FUNCTION_BLOCK FB_ModbusCon
VAR_INPUT
    bEnable: BOOL;
END_VAR
VAR_OUTPUT
    // Operating data from inverter
    stInverter: ST_OpDataInverter;
    // Operating data from meter
    stMeter: ST_OpDataMeter;
    // Operating data from storage
    stStorage: ST_OpDataStorage;
    // Connection is ready and not locked out
    bReady: BOOL;
END_VAR
VAR
    // IP address of the target device
    {attribute 'hide'}
    _sInverterIPAddr: STRING;
    // Port number of the target device
    {attribute 'hide'}
    _nInverterTCPPort: UINT;
    // Modbus RTU ID of inverter, value must be 16#FF if addressed directly via TCP/IP
    {attribute 'hide'}
    _nInverterUnitID: BYTE;
    // Modbus RTU ID of meter, value must be 16#FF if addressed directly via TCP/IP
    {attribute 'hide'}
    _nMeterUnitID: BYTE;
    // Timeout that may not be exceeded by execution of the ADS command
    {attribute 'hide'}
    _tConnectionTimeout: TIME;
    // Timeout between modbus commands sent to target device
    {attribute 'hide'}
    _tConnectionCoolDown: TIME;

    // Modbus connection to read registers
    fbReadRegister: FB_MBReadRegs;
    // Connection cooldown timeout between requests
    fbConnectionCoolDown: TOF;

    // Register data of inverter
    stInverterRegisterData: ST_RegMapInverter;
    // Register data of meter
    stMeterRegisterData: ST_RegMapMeter;
    // Register data of storage
    stStorageRegisterData: ST_RegMapStorage;

    // Number of current tried countermeasures after modbus connection error
    nConnectionCountermeasure: INT;
    // Number of current tried countermeasures after modbus request error regarding inverter
    nInverterCountermeasure: INT;
    // Number of current tried countermeasures after modbus request error regarding meter
    nMeterCountermeasure: INT;
    // Number of current tried countermeasures after modbus request error regarding storage
    nStorageCountermeasure: INT;

    // Current state of modbus read registers
    eReadState: (WAIT_FOR_ENABLE, PREPARE_READ_REGS, EXECUTE_READ_REGS, WAIT_READ_REGS_FEEDBACK, ASSIGN_VALUES, SELECT_NEXT_SUBSYTEM, CON_COOL_DOWN, CON_LOCKOUT);
    // Select subsystem for request to prevent parallel requests
    eCurrentSubsystem: (INVERTER, METER, STORAGE);

    // Show only events with minimum severety level
    {attribute 'hide'}
    _eTraceLevel: TcEventSeverity := TcEventSeverity.Warning;

    fbAlarmMbConnectionError: FB_TcAlarm;
    fbAlarmMbFunctionInverterError: FB_TcAlarm;
    fbAlarmMbFunctionMeterError: FB_TcAlarm;
    fbAlarmMbFunctionStorageError: FB_TcAlarm;
    fbAlarmMbConnectionLocked: FB_TcAlarm;
    fbMessageMbOpDataIsUpdated: FB_TcMessage;
    fbMessageMbUncatchedError: FB_TcMessage;
    fbMessageMbReceivedBytesMismatch: FB_TcMessage;
END_VAR
VAR CONSTANT
    // Number of output registers used by stInverterRegisterData
    nInverterRegQuantity: WORD := 16;
    // Start address of the output register used by stInverterRegisterData
    nInverterMBStartAddr: WORD := 40071;
    // Number of output registers used by stMeterRegisterData
    nMeterRegQuantity: WORD := 21;
    // Start address of the output register used by stMeterRegisterData
    nMeterMBStartAddr: WORD := 40071;
    // Number of output registers used by stStorageRegisterData
    nStorageRegQuantity: WORD := 4;
    // Start address of the output register used by stStorageRegisterData
    nStorageMBStartAddr: WORD := 40351;
    // Number of attempted countermeasures before connection lockout (connection error)
    nConnectionCmBeforeLockout: INT := 5;
    // Number of attempted countermeasures before connection lockout (subsystem error)
    nSubsystemCmBeforeLockout: INT := 2;
END_VAR

fbReadRegister(sIPAddr := sInverterIPAddr, nTCPPort := nInverterTCPPort, tTimeout := tConnectionTimeout);
fbConnectionCoolDown();

// Set ready state
bReady := eReadState <> CON_LOCKOUT;

// Default operating data has not been updated this cycle
stInverter.bOpDataIsUpdated := FALSE;
stMeter.bOpDataIsUpdated := FALSE;
stStorage.bOpDataIsUpdated := FALSE;

// State machine
CASE eReadState OF
    WAIT_FOR_ENABLE:
        IF bEnable AND fbConnectionCoolDown.Q THEN
            eReadState := CON_COOL_DOWN;
        ELSIF bEnable THEN
            eReadState := PREPARE_READ_REGS;
        END_IF

    PREPARE_READ_REGS:
        CASE eCurrentSubsystem OF
            INVERTER:
                fbReadRegister.nUnitID := nInverterUnitID;
                fbReadRegister.nQuantity := nInverterRegQuantity;
                fbReadRegister.nMBAddr := nInverterMBStartAddr;
                fbReadRegister.cbLength := SIZEOF(stInverterRegisterData);
                fbReadRegister.pDestAddr := ADR(stInverterRegisterData);

            METER:
                fbReadRegister.nUnitID := nMeterUnitID;
                fbReadRegister.nQuantity := nMeterRegQuantity;
                fbReadRegister.nMBAddr := nMeterMBStartAddr;
                fbReadRegister.cbLength := SIZEOF(stMeterRegisterData);
                fbReadRegister.pDestAddr := ADR(stMeterRegisterData);

            STORAGE:
                fbReadRegister.nUnitID := nInverterUnitID;
                fbReadRegister.nQuantity := nStorageRegQuantity;
                fbReadRegister.nMBAddr := nStorageMBStartAddr;
                fbReadRegister.cbLength := SIZEOF(stStorageRegisterData) - 2;
                fbReadRegister.pDestAddr := ADR(stStorageRegisterData);
        END_CASE

        eReadState := EXECUTE_READ_REGS;

    EXECUTE_READ_REGS:
        fbReadRegister.bExecute := TRUE;
        fbConnectionCoolDown.IN := TRUE;
        eReadState := WAIT_READ_REGS_FEEDBACK;

    WAIT_READ_REGS_FEEDBACK:
        fbReadRegister.bExecute := FALSE;
        IF NOT fbReadRegister.bBusy THEN
            fbConnectionCoolDown.IN := FALSE;
            ConnectionErrorHandler();

            IF ConnectionLockoutIsActive() THEN
                // Lockout modbus connection
                eReadState := CON_LOCKOUT;
            ELSIF fbReadRegister.cbLength <> fbReadRegister.cbRead THEN
                // Send message M_MbReceivedBytesMismatch
                IF fbMessageMbReceivedBytesMismatch.eSeverity >= eTraceLevel THEN
                    fbMessageMbReceivedBytesMismatch.ipArguments.Clear();
                    fbMessageMbReceivedBytesMismatch.ipArguments.AddBool(value := eCurrentSubsystem = INVERTER);
                    fbMessageMbReceivedBytesMismatch.ipArguments.AddBool(value := eCurrentSubsystem = METER);
                    fbMessageMbReceivedBytesMismatch.ipArguments.AddBool(value := eCurrentSubsystem = STORAGE);
                    fbMessageMbReceivedBytesMismatch.Send();
                END_IF
                // Skip assigning values to output variable
                eReadState := SELECT_NEXT_SUBSYTEM;
            ELSE
                eReadState := ASSIGN_VALUES;
            END_IF
        END_IF

    ASSIGN_VALUES:
        CASE eCurrentSubsystem OF
            INVERTER:
                stInverter.bOpDataIsUpdated := TRUE;
                stInverter.fCurrentL1 := Scale(stInverterRegisterData.nCurrentL1, stInverterRegisterData.nSfCurrent);
                stInverter.fCurrentL2 := Scale(stInverterRegisterData.nCurrentL2, stInverterRegisterData.nSfCurrent);
                stInverter.fCurrentL3 := Scale(stInverterRegisterData.nCurrentL3, stInverterRegisterData.nSfCurrent);
                stInverter.fVoltageL1L2 := Scale(stInverterRegisterData.nVoltageL1L2, stInverterRegisterData.nSfVoltage);
                stInverter.fVoltageL2L3 := Scale(stInverterRegisterData.nVoltageL2L3, stInverterRegisterData.nSfVoltage);
                stInverter.fVoltageL3L1 := Scale(stInverterRegisterData.nVoltageL3L1, stInverterRegisterData.nSfVoltage);
                stInverter.fVoltageL1N := Scale(stInverterRegisterData.nVoltageL1N, stInverterRegisterData.nSfVoltage);
                stInverter.fVoltageL2N := Scale(stInverterRegisterData.nVoltageL2N, stInverterRegisterData.nSfVoltage);
                stInverter.fVoltageL3N := Scale(stInverterRegisterData.nVoltageL3N, stInverterRegisterData.nSfVoltage);
                stInverter.fPower := Scale(stInverterRegisterData.nPower, stInverterRegisterData.nSfPower);
                stInverter.fFrequency := Scale(stInverterRegisterData.nFrequency, stInverterRegisterData.nSfFrequency);

            METER:
                stMeter.bOpDataIsUpdated := TRUE;
                stMeter.fCurrentL1 := Scale(stMeterRegisterData.nCurrentL1, stMeterRegisterData.nSfCurrent);
                stMeter.fCurrentL2 := Scale(stMeterRegisterData.nCurrentL2, stMeterRegisterData.nSfCurrent);
                stMeter.fCurrentL3 := Scale(stMeterRegisterData.nCurrentL3, stMeterRegisterData.nSfCurrent);
                stMeter.fVoltageL1L2 := Scale(stMeterRegisterData.nVoltageL1L2, stMeterRegisterData.nSfVoltage);
                stMeter.fVoltageL2L3 := Scale(stMeterRegisterData.nVoltageL2L3, stMeterRegisterData.nSfVoltage);
                stMeter.fVoltageL3L1 := Scale(stMeterRegisterData.nVoltageL3L1, stMeterRegisterData.nSfVoltage);
                stMeter.fVoltageL1N := Scale(stMeterRegisterData.nVoltageL1N, stMeterRegisterData.nSfVoltage);
                stMeter.fVoltageL2N := Scale(stMeterRegisterData.nVoltageL2N, stMeterRegisterData.nSfVoltage);
                stMeter.fVoltageL3N := Scale(stMeterRegisterData.nVoltageL3N, stMeterRegisterData.nSfVoltage);
                stMeter.fPower := Scale(stMeterRegisterData.nPower, stMeterRegisterData.nSfPower);
                stMeter.fPowerL1 := Scale(stMeterRegisterData.nPowerL1, stMeterRegisterData.nSfPower) - 100;
                stMeter.fPowerL2 := Scale(stMeterRegisterData.nPowerL2, stMeterRegisterData.nSfPower) - 100;
                stMeter.fPowerL3 := Scale(stMeterRegisterData.nPowerL3, stMeterRegisterData.nSfPower) - 100;
                stMeter.fFrequency := Scale(stMeterRegisterData.nFrequency, stMeterRegisterData.nSfFrequency);

            STORAGE:
                stStorage.bOpDataIsUpdated := TRUE;
                stStorage.nStateOfCharge := REAL_TO_INT(Scale(stStorageRegisterData.nStateOfCharge, stStorageRegisterData.nSfStateOfCharge));
                stStorage.eState := stStorageRegisterData.nState;
        END_CASE
        eReadState := SELECT_NEXT_SUBSYTEM;

        // Send message M_MbOpDataIsUpdated
        IF fbMessageMbOpDataIsUpdated.eSeverity >= eTraceLevel THEN
            fbMessageMbOpDataIsUpdated.ipArguments.Clear();
            fbMessageMbOpDataIsUpdated.ipArguments.AddBool(value := stInverter.bOpDataIsUpdated);
            fbMessageMbOpDataIsUpdated.ipArguments.AddBool(value := stMeter.bOpDataIsUpdated);
            fbMessageMbOpDataIsUpdated.ipArguments.AddBool(value := stStorage.bOpDataIsUpdated);
            fbMessageMbOpDataIsUpdated.Send();
        END_IF

    SELECT_NEXT_SUBSYTEM:
        CASE eCurrentSubsystem OF
            INVERTER:
                eCurrentSubsystem := METER;

            METER:
                eCurrentSubsystem := STORAGE;

            STORAGE:
                eCurrentSubsystem := INVERTER;

            ELSE
                eCurrentSubsystem := INVERTER;
        END_CASE
        eReadState := CON_COOL_DOWN;

    CON_COOL_DOWN:
        IF NOT bEnable THEN
            eReadState := WAIT_FOR_ENABLE;
        END_IF

        IF NOT fbConnectionCoolDown.Q THEN
            eReadState := PREPARE_READ_REGS;
        END_IF

    CON_LOCKOUT:
        (* Perform reset using Reset() function *)
END_CASE

METHOD PRIVATE ConnectionErrorHandler
IF ConnectionLockoutIsActive() THEN
    RETURN;
END_IF

IF fbReadRegister.bError THEN
    // Apply countermeasure if ADS error occured
    CASE fbReadRegister.nErrId OF
        16#8001, // Modbus function not implemented
        16#8002, // Invalid address or length
        16#8003, // Invalid parameters: incorrect number of registers
        16#8004: // Modbus server error
            CASE eCurrentSubsystem OF
                INVERTER:
                    nInverterCountermeasure := nInverterCountermeasure + 1;
                METER:
                    nMeterCountermeasure := nMeterCountermeasure + 1;
                STORAGE:
                    nStorageCountermeasure := nStorageCountermeasure + 1;
            END_CASE
            

        Global.E_TcSystemEventClass.TCPSendError, // TCP send error
        Tc2_System.E_AdsErr.CLIENT_SYNCTIMEOUT:   // Remote terminal is not responding in the specified ADS timeout
            nConnectionCountermeasure := nConnectionCountermeasure + 1;
            fbConnectionCoolDown.PT := tConnectionCoolDown + tConnectionCoolDown * LREAL_TO_INT(EXPT(nConnectionCountermeasure, 2));

        ELSE
            // Send message M_MbUncatchedError
            IF fbMessageMbUncatchedError.eSeverity >= eTraceLevel THEN
                fbMessageMbUncatchedError.ipArguments.Clear();
                fbMessageMbUncatchedError.ipArguments.AddUDInt(value := fbReadRegister.nErrId);
                fbMessageMbUncatchedError.Send();
            END_IF
    END_CASE

ELSE
    // Defer possibly still active countermeasure
    nInverterCountermeasure := 0;
    nMeterCountermeasure := 0;
    nStorageCountermeasure := 0;
    nConnectionCountermeasure := 0;

    // Reset connection cooldown timeout
    fbConnectionCoolDown.PT := tConnectionCoolDown;
END_IF

IF nConnectionCountermeasure > 0 AND fbAlarmMbConnectionError.eSeverity >= eTraceLevel AND NOT fbAlarmMbConnectionError.bRaised THEN
    // Raise alarm F_MbConnectionError
    fbAlarmMbConnectionError.ipArguments.AddUDInt(value := fbReadRegister.nErrId);
    fbAlarmMbConnectionError.Raise();
ELSIF nConnectionCountermeasure = 0 AND fbAlarmMbConnectionError.bRaised THEN
    // Clear alarm F_MbConnectionError
    fbAlarmMbConnectionError.ipArguments.Clear();
    fbAlarmMbConnectionError.Clear();
END_IF

IF nInverterCountermeasure > 0 AND fbAlarmMbFunctionInverterError.eSeverity >= eTraceLevel AND NOT fbAlarmMbFunctionInverterError.bRaised THEN
    // Raise alarm F_MbFunctionInverterError
    fbAlarmMbFunctionInverterError.ipArguments.AddUDInt(value := fbReadRegister.nErrId);
    fbAlarmMbFunctionInverterError.Raise();
ELSIF nInverterCountermeasure = 0 AND fbAlarmMbFunctionInverterError.bRaised THEN
    // Clear alarm F_MbFunctionInverterError
    fbAlarmMbFunctionInverterError.ipArguments.Clear();
    fbAlarmMbFunctionInverterError.Clear();
END_IF

IF nMeterCountermeasure > 0 AND fbAlarmMbFunctionMeterError.eSeverity >= eTraceLevel AND NOT fbAlarmMbFunctionMeterError.bRaised THEN
    // Raise alarm F_MbFunctionMeterError
    fbAlarmMbFunctionMeterError.ipArguments.AddUDInt(value := fbReadRegister.nErrId);
    fbAlarmMbFunctionMeterError.Raise();
ELSIF nMeterCountermeasure = 0 AND fbAlarmMbFunctionMeterError.bRaised THEN
    // Clear alarm F_MbFunctionMeterError
    fbAlarmMbFunctionMeterError.ipArguments.Clear();
    fbAlarmMbFunctionMeterError.Clear();
END_IF

IF nStorageCountermeasure > 0 AND fbAlarmMbFunctionStorageError.eSeverity >= eTraceLevel AND NOT fbAlarmMbFunctionStorageError.bRaised THEN
    // Raise alarm F_MbFunctionStorageError
    fbAlarmMbFunctionStorageError.ipArguments.AddUDInt(value := fbReadRegister.nErrId);
    fbAlarmMbFunctionStorageError.Raise();
ELSIF nStorageCountermeasure = 0 AND fbAlarmMbFunctionStorageError.bRaised THEN
    // Clear alarm F_MbFunctionStorageError
    fbAlarmMbFunctionStorageError.ipArguments.Clear();
    fbAlarmMbFunctionStorageError.Clear();
END_IF
END_METHOD

METHOD PRIVATE ConnectionLockoutIsActive : BOOL
// Default to false, no lockout active
ConnectionLockoutIsActive := FALSE;

// Return if already in locked state
IF eReadState = CON_LOCKOUT THEN
    ConnectionLockoutIsActive := TRUE;
    RETURN;
END_IF

IF nConnectionCountermeasure > nConnectionCmBeforeLockout THEN
    ConnectionLockoutIsActive := TRUE;
    // Add reference to F_MbConnectionError as argument to F_MbConnectionLocked
    IF fbAlarmMbConnectionLocked.eSeverity >= eTraceLevel AND NOT fbAlarmMbConnectionLocked.bRaised THEN
        fbAlarmMbConnectionLocked.ipArguments.AddEventReferenceId(nEventId := fbAlarmMbConnectionError.nEventId);
    END_IF
END_IF

if nInverterCountermeasure > nSubsystemCmBeforeLockout THEN
    ConnectionLockoutIsActive := TRUE;
    // Add reference to F_MbFunctionInverterError as argument to F_MbConnectionLocked
    IF fbAlarmMbConnectionLocked.eSeverity >= eTraceLevel AND NOT fbAlarmMbConnectionLocked.bRaised THEN
        fbAlarmMbConnectionLocked.ipArguments.AddEventReferenceId(nEventId := fbAlarmMbFunctionInverterError.nEventId);
    END_IF
END_IF

if nMeterCountermeasure > nSubsystemCmBeforeLockout THEN
    ConnectionLockoutIsActive := TRUE;
    // Add reference to F_MbFunctionMeterError as argument to F_MbConnectionLocked
    IF fbAlarmMbConnectionLocked.eSeverity >= eTraceLevel AND NOT fbAlarmMbConnectionLocked.bRaised THEN
        fbAlarmMbConnectionLocked.ipArguments.AddEventReferenceId(nEventId := fbAlarmMbFunctionMeterError.nEventId);
    END_IF
END_IF

if nStorageCountermeasure > nSubsystemCmBeforeLockout THEN
    ConnectionLockoutIsActive := TRUE;
    // Add reference to F_MbFunctionStorageError as argument to F_MbConnectionLocked
    IF fbAlarmMbConnectionLocked.eSeverity >= eTraceLevel AND NOT fbAlarmMbConnectionLocked.bRaised THEN
        fbAlarmMbConnectionLocked.ipArguments.AddEventReferenceId(nEventId := fbAlarmMbFunctionStorageError.nEventId);
    END_IF
END_IF

IF ConnectionLockoutIsActive AND fbAlarmMbConnectionLocked.eSeverity >= eTraceLevel AND NOT fbAlarmMbConnectionLocked.bRaised THEN
    // Raise alarm F_MbConnectionLocked
    fbAlarmMbConnectionLocked.Raise();
END_IF
END_METHOD

// Show only events with minimum severety level
{attribute 'monitoring' := 'call'}
PROPERTY eTraceLevel : Global.TcEventSeverity
GET
eTraceLevel := _eTraceLevel;
END_GET
SET
_eTraceLevel := eTraceLevel;
END_SET
END_PROPERTY

METHOD FB_Init: BOOL
VAR_INPUT
    // TRUE: the retain variables are initialized (reset warm / reset cold)
    bInitRetains: BOOL;
    // TRUE: the instance will be copied to the copy code afterward (online change)      
    bInCopyCode: BOOL; 
END_VAR
// Create alarm/message instances for the event logger
IF NOT bInCopyCode THEN
    fbAlarmMbConnectionError.CreateEx(stEventEntry := TC_EVENTS.MainControllerEventClass.F_MbConnectionError, bWithConfirmation := FALSE);
    fbAlarmMbFunctionInverterError.CreateEx(stEventEntry := TC_EVENTS.MainControllerEventClass.F_MbFunctionInverterError, bWithConfirmation := FALSE);
    fbAlarmMbFunctionMeterError.CreateEx(stEventEntry := TC_EVENTS.MainControllerEventClass.F_MbFunctionMeterError, bWithConfirmation := FALSE);
    fbAlarmMbFunctionStorageError.CreateEx(stEventEntry := TC_EVENTS.MainControllerEventClass.F_MbFunctionStorageError, bWithConfirmation := FALSE);
    fbAlarmMbConnectionLocked.CreateEx(stEventEntry := TC_EVENTS.MainControllerEventClass.F_MbConnectionLocked, bWithConfirmation := FALSE);
    fbMessageMbOpDataIsUpdated.CreateEx(stEventEntry := TC_EVENTS.MainControllerEventClass.M_MbOpDataIsUpdated);
    fbMessageMbUncatchedError.CreateEx(stEventEntry := TC_EVENTS.MainControllerEventClass.M_MbUncatchedError);
    fbMessageMbReceivedBytesMismatch.CreateEx(stEventEntry := TC_EVENTS.MainControllerEventClass.M_MbReceivedBytesMismatch);
END_IF
END_METHOD

// IP address of the target device
{attribute 'monitoring' := 'variable'}
PROPERTY nInverterTCPPort : UINT
GET
nInverterTCPPort := _nInverterTCPPort;
END_GET
SET
_nInverterTCPPort := nInverterTCPPort;
END_SET
END_PROPERTY

// Modbus RTU ID of inverter, value must be 16#FF if addressed directly via TCP/IP
{attribute 'monitoring' := 'variable'}
PROPERTY nInverterUnitID : BYTE
GET
nInverterUnitID := _nInverterUnitID;
END_GET
SET
_nInverterUnitID := nInverterUnitID;
END_SET
END_PROPERTY

// Modbus RTU ID of meter, value must be 16#FF if addressed directly via TCP/IP
{attribute 'monitoring' := 'variable'}
PROPERTY nMeterUnitID : BYTE
GET
nMeterUnitID := _nMeterUnitID;
END_GET
SET
_nMeterUnitID := nMeterUnitID;
END_SET
END_PROPERTY

METHOD PUBLIC Reset
nInverterCountermeasure := 0;
nMeterCountermeasure := 0;
nStorageCountermeasure := 0;
nConnectionCountermeasure := 0;

eReadState := WAIT_FOR_ENABLE;

// Clear alarm F_MbConnectionLocked
fbAlarmMbConnectionLocked.Clear();
fbAlarmMbConnectionLocked.ipArguments.Clear();
END_METHOD

METHOD PRIVATE Scale : REAL
VAR_INPUT
    nValue: WORD;
    nScaleFactor: WORD;
END_VAR
Scale := nValue * LREAL_TO_REAL(EXPT(10, UINT_TO_INT(nScaleFactor)));
END_METHOD

// IP address of the target device
{attribute 'monitoring' := 'variable'}
PROPERTY sInverterIPAddr : STRING
GET
sInverterIPAddr := _sInverterIPAddr;
END_GET
SET
_sInverterIPAddr := sInverterIPAddr;
END_SET
END_PROPERTY

// Timeout between modbus commands sent to target device
{attribute 'monitoring' := 'call'}
PROPERTY tConnectionCoolDown : TIME
GET
tConnectionCoolDown := _tConnectionCoolDown;
END_GET
SET
_tConnectionCoolDown := tConnectionCoolDown;

// Apply connection cooldown timeout if no counter measure is active
IF nConnectionCountermeasure = 0 AND nInverterCountermeasure = 0 AND nMeterCountermeasure = 0 AND nStorageCountermeasure = 0 THEN
    fbConnectionCoolDown.PT := tConnectionCoolDown;
END_IF
END_SET
END_PROPERTY

// Timeout that may not be exceeded by execution of the ADS command
{attribute 'monitoring' := 'call'}
PROPERTY tConnectionTimeout : TIME
GET
tConnectionTimeout := _tConnectionTimeout;
END_GET
SET
_tConnectionTimeout := tConnectionTimeout;
END_SET
END_PROPERTY

END_FUNCTION_BLOCK

(* stored: Version 1.1.0.1
   POU FB_ModbusCon: Id {43065017-eb91-4d51-b9c6-b54abe313361}, SpecialFunc None
   Folder Properties: Id {e526952d-1a01-4e02-a2fb-614c560a061a}
   Method ConnectionErrorHandler: Id {eb35efc9-f4bd-48ca-9579-f04d9ee594f3}
   Method ConnectionLockoutIsActive: Id {bf05b0a2-a100-4785-9923-1a19614766ee}
   Property eTraceLevel: Id {18801b62-0a1d-4b15-a681-6dc568dda570}
   Get Get: Id {151d98d5-adff-4121-9726-572ac2cfec04}
   Set Set: Id {b3395472-f3ef-4c16-9a44-b0aedb84921e}
   Method FB_Init: Id {d1de6e2a-f58c-4b67-ae69-3ec139555bef}
   Property nInverterTCPPort: Id {0208614e-59f7-4633-83e9-f19d97c40446}
   Get Get: Id {0751807e-b515-449a-81b0-294d4ae71c2d}
   Set Set: Id {73510e41-675d-4b24-b148-178637450bd3}
   Property nInverterUnitID: Id {4b091f00-d0cf-42a0-8a80-698bd7c0cb80}
   Get Get: Id {203f77d2-9bd0-44e9-b1f5-d0e6a98b84c1}
   Set Set: Id {13d50004-a553-4bfb-a6c8-e2e4794064b3}
   Property nMeterUnitID: Id {527b1d04-a12e-4bee-93ec-d9b28a6a9926}
   Get Get: Id {a4b3b186-664a-4b6a-ac57-3ad93c32bb74}
   Set Set: Id {3c2feef1-2f4b-477a-b581-ec4705605620}
   Method Reset: Id {dcc751c1-95e6-4506-87cb-37fdf657bcaf}
   Method Scale: Id {42cdecb6-346c-42d7-8d00-085967a56f85}
   Property sInverterIPAddr: Id {bb6c70b4-566d-44aa-9bf4-f7634820c67a}
   Get Get: Id {898b2f55-6363-49f6-b4cc-12a33e04db4b}
   Set Set: Id {c27586e5-8cd9-4e3e-ac15-5a3ff0e940de}
   Property tConnectionCoolDown: Id {6f8307c1-4b4e-402e-9adb-89621f0deb8a}
   Get Get: Id {7e0cee8a-5fc2-457f-8bf4-bf2545934b94}
   Set Set: Id {a4cab1d9-c121-4bcb-a3ec-859f2ad4656e}
   Property tConnectionTimeout: Id {e5048373-5545-4343-bd36-b4a6dfb3f32d}
   Get Get: Id {1a2f3e9b-eb8a-4180-b874-494a0b9ca5aa}
   Set Set: Id {afb1dd33-6454-4ce6-a3e7-ff21ccd34cf4} *)
